// LS Electric XG5000 project: 과년65_1
// PLC NewPLC
// module base 0 slot 0: 입출력 모듈:XBC-DR20S (DC 24V 입력 12점, 릴레이 출력 8점)

PROGRAM NewProgram (task: 스캔 프로그램)

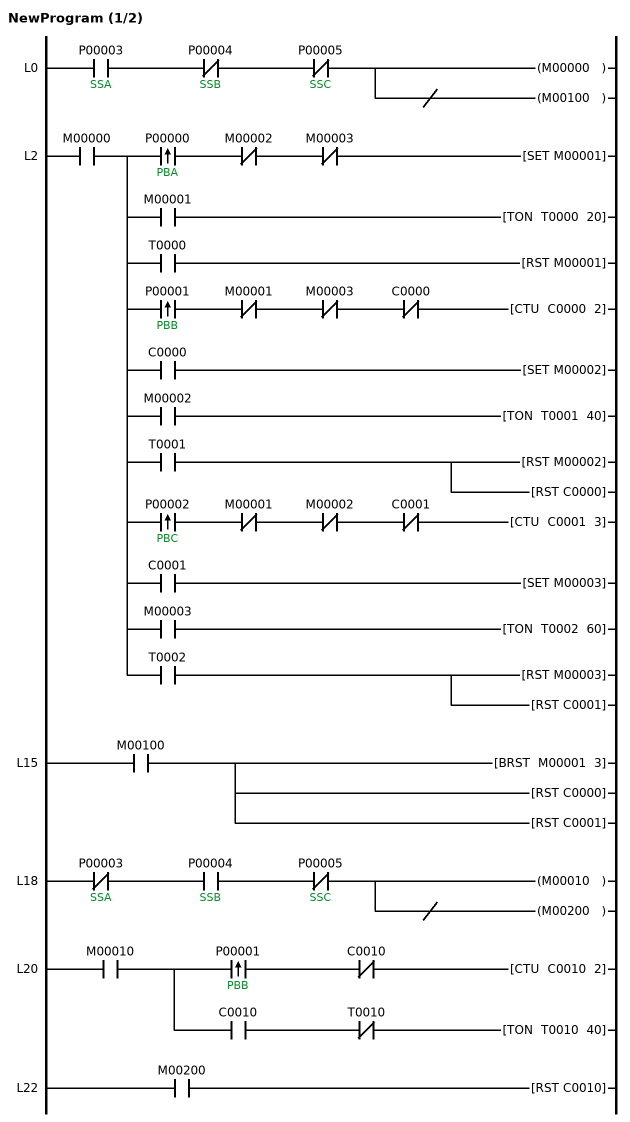
; L0
LOAD      P00003	// SSA
AND NOT   P00004	// SSB
AND NOT   P00005	// SSC
OUT       M00000
NOT
OUT       M00100
; L2
LOAD      M00000
MPUSH
ANDP      P00000	// PBA
AND NOT   M00002
AND NOT   M00003
SET       M00001
MLOAD
AND       M00001
TON       T0000 20
MLOAD
AND       T0000
RST       M00001
MLOAD
ANDP      P00001	// PBB
AND NOT   M00001
AND NOT   M00003
AND NOT   C0000
CTU       C0000 2
MLOAD
AND       C0000
SET       M00002
MLOAD
AND       M00002
TON       T0001 40
MLOAD
AND       T0001
RST       M00002
RST       C0000
MLOAD
ANDP      P00002	// PBC
AND NOT   M00001
AND NOT   M00002
AND NOT   C0001
CTU       C0001 3
MLOAD
AND       C0001
SET       M00003
MLOAD
AND       M00003
TON       T0002 60
MPOP
AND       T0002
RST       M00003
RST       C0001
; L15
LOAD      M00100
BRST      M00001 3
RST       C0000
RST       C0001
; L18
LOAD NOT  P00003	// SSA
AND       P00004	// SSB
AND NOT   P00005	// SSC
OUT       M00010
NOT
OUT       M00200
; L20
LOAD      M00010
MPUSH
ANDP      P00001	// PBB
AND NOT   C0010
CTU       C0010 2
MPOP
AND       C0010
AND NOT   T0010
TON       T0010 40
; L22
LOAD      M00200
RST       C0010

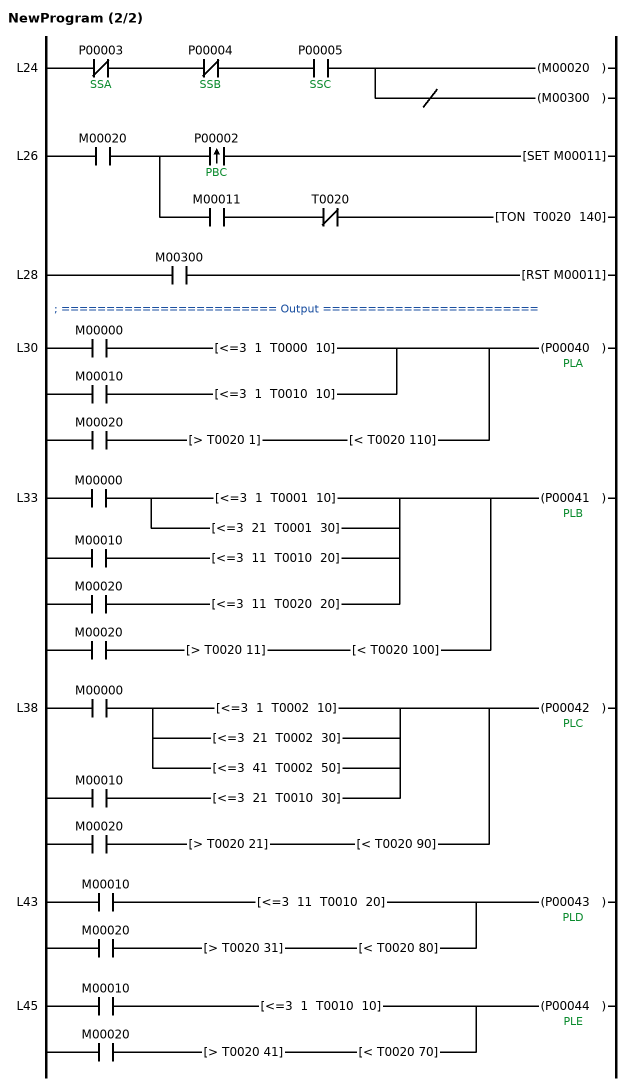
; L24
LOAD NOT  P00003	// SSA
AND NOT   P00004	// SSB
AND       P00005	// SSC
OUT       M00020
NOT
OUT       M00300
; L26
LOAD      M00020
MPUSH
ANDP      P00002	// PBC
SET       M00011
MPOP
AND       M00011
AND NOT   T0020
TON       T0020 140
; L28
LOAD      M00300
RST       M00011
// ======================== Output ========================
; L30
LOAD      M00000
AND<=3    1 T0000 10
LOAD      M00010
AND<=3    1 T0010 10
OR LOAD
LOAD      M00020
AND>      T0020 1
AND<      T0020 110
OR LOAD
OUT       P00040	// PLA
; L33
LOAD      M00000
LOAD<=3   1 T0001 10
OR<=3     21 T0001 30
AND LOAD
LOAD      M00010
AND<=3    11 T0010 20
OR LOAD
LOAD      M00020
AND<=3    11 T0020 20
OR LOAD
LOAD      M00020
AND>      T0020 11
AND<      T0020 100
OR LOAD
OUT       P00041	// PLB
; L38
LOAD      M00000
LOAD<=3   1 T0002 10
OR<=3     21 T0002 30
OR<=3     41 T0002 50
AND LOAD
LOAD      M00010
AND<=3    21 T0010 30
OR LOAD
LOAD      M00020
AND>      T0020 21
AND<      T0020 90
OR LOAD
OUT       P00042	// PLC
; L43
LOAD      M00010
AND<=3    11 T0010 20
LOAD      M00020
AND>      T0020 31
AND<      T0020 80
OR LOAD
OUT       P00043	// PLD
; L45
LOAD      M00010
AND<=3    1 T0010 10
LOAD      M00020
AND>      T0020 41
AND<      T0020 70
OR LOAD
OUT       P00044	// PLE